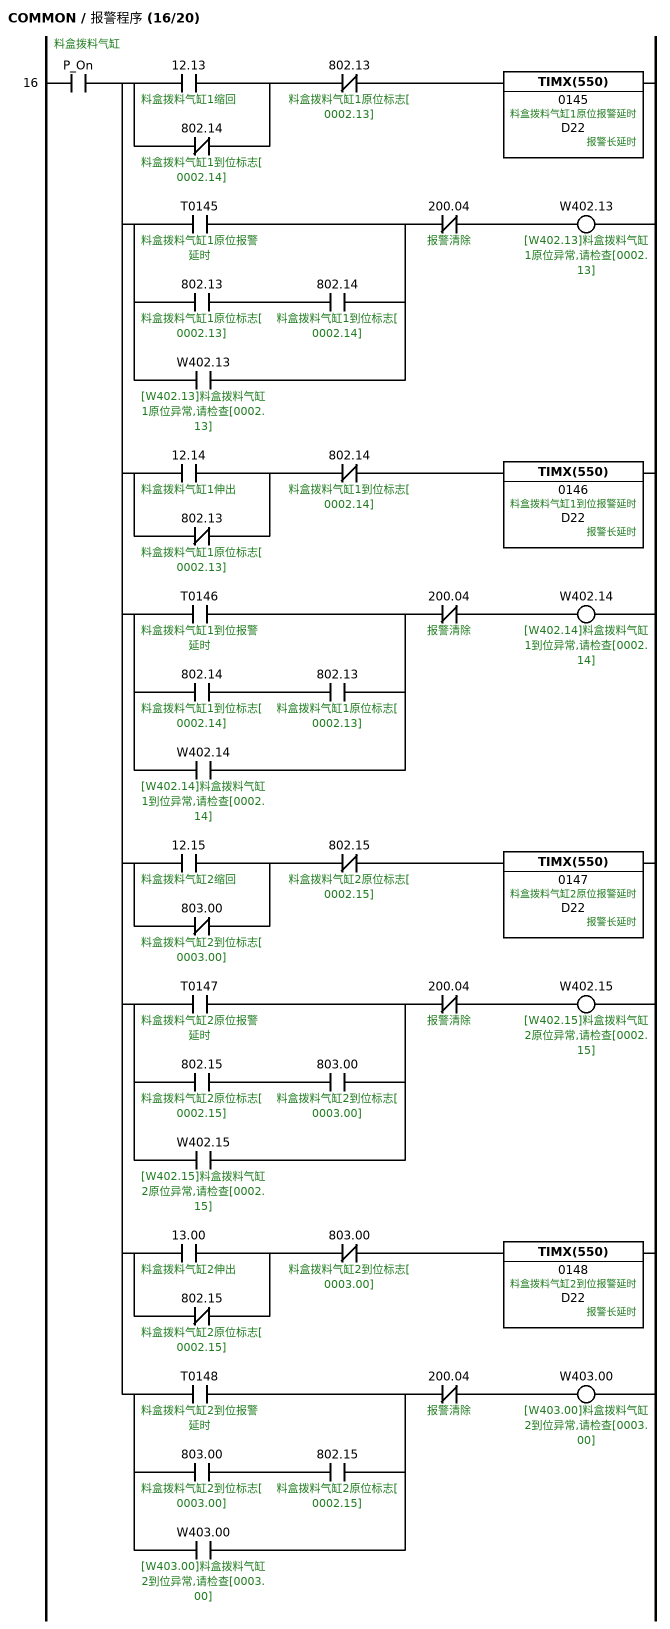
; [picture p192: COMMON / 报警程序, rungs 16-16]
; rung 16: 料盒拨料气缸
LD P_On
OUT TR0
LD 12.13  ; 料盒拨料气缸1缩回
ORNOT 802.14  ; 料盒拨料气缸1到位标志[0002.14]
ANDLD
ANDNOT 802.13  ; 料盒拨料气缸1原位标志[0002.13]
TIMX(550) 0145 D22  ; 报警长延时, 料盒拨料气缸1原位报警延时
LD TR0
LD T0145  ; 料盒拨料气缸1原位报警延时
LD 802.13  ; 料盒拨料气缸1原位标志[0002.13]
AND 802.14  ; 料盒拨料气缸1到位标志[0002.14]
ORLD
OR W402.13  ; [W402.13]料盒拨料气缸1原位异常,请检查[0002.13]
ANDLD
ANDNOT 200.04  ; 报警清除
OUT W402.13  ; [W402.13]料盒拨料气缸1原位异常,请检查[0002.13]
LD TR0
LD 12.14  ; 料盒拨料气缸1伸出
ORNOT 802.13  ; 料盒拨料气缸1原位标志[0002.13]
ANDLD
ANDNOT 802.14  ; 料盒拨料气缸1到位标志[0002.14]
TIMX(550) 0146 D22  ; 报警长延时, 料盒拨料气缸1到位报警延时
LD TR0
LD T0146  ; 料盒拨料气缸1到位报警延时
LD 802.14  ; 料盒拨料气缸1到位标志[0002.14]
AND 802.13  ; 料盒拨料气缸1原位标志[0002.13]
ORLD
OR W402.14  ; [W402.14]料盒拨料气缸1到位异常,请检查[0002.14]
ANDLD
ANDNOT 200.04  ; 报警清除
OUT W402.14  ; [W402.14]料盒拨料气缸1到位异常,请检查[0002.14]
LD TR0
LD 12.15  ; 料盒拨料气缸2缩回
ORNOT 803.00  ; 料盒拨料气缸2到位标志[0003.00]
ANDLD
ANDNOT 802.15  ; 料盒拨料气缸2原位标志[0002.15]
TIMX(550) 0147 D22  ; 报警长延时, 料盒拨料气缸2原位报警延时
LD TR0
LD T0147  ; 料盒拨料气缸2原位报警延时
LD 802.15  ; 料盒拨料气缸2原位标志[0002.15]
AND 803.00  ; 料盒拨料气缸2到位标志[0003.00]
ORLD
OR W402.15  ; [W402.15]料盒拨料气缸2原位异常,请检查[0002.15]
ANDLD
ANDNOT 200.04  ; 报警清除
OUT W402.15  ; [W402.15]料盒拨料气缸2原位异常,请检查[0002.15]
LD TR0
LD 13.00  ; 料盒拨料气缸2伸出
ORNOT 802.15  ; 料盒拨料气缸2原位标志[0002.15]
ANDLD
ANDNOT 803.00  ; 料盒拨料气缸2到位标志[0003.00]
TIMX(550) 0148 D22  ; 报警长延时, 料盒拨料气缸2到位报警延时
LD TR0
LD T0148  ; 料盒拨料气缸2到位报警延时
LD 803.00  ; 料盒拨料气缸2到位标志[0003.00]
AND 802.15  ; 料盒拨料气缸2原位标志[0002.15]
ORLD
OR W403.00  ; [W403.00]料盒拨料气缸2到位异常,请检查[0003.00]
ANDLD
ANDNOT 200.04  ; 报警清除
OUT W403.00  ; [W403.00]料盒拨料气缸2到位异常,请检查[0003.00]

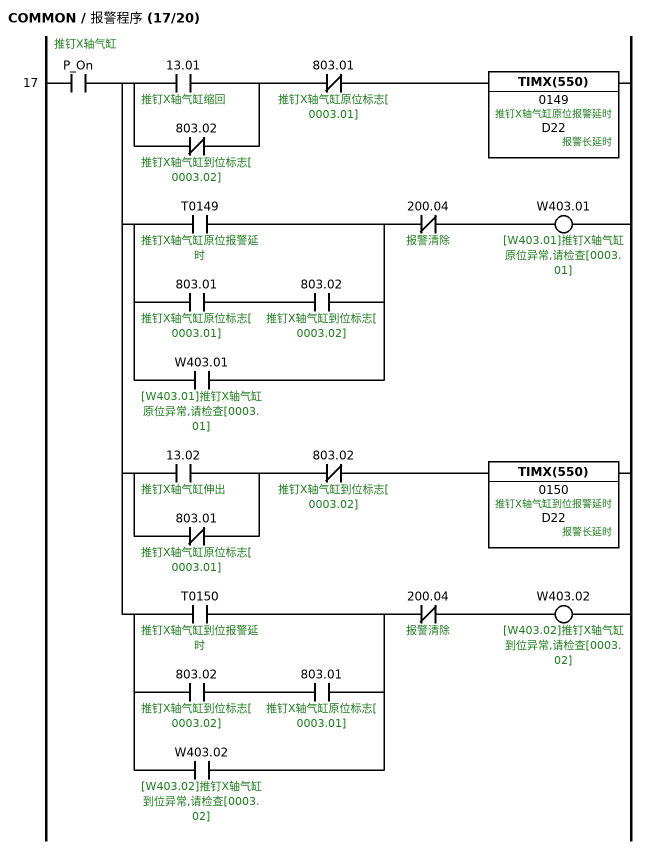
; rung 17: 推钉X轴气缸
LD P_On
OUT TR0
LD 13.01  ; 推钉X轴气缸缩回
ORNOT 803.02  ; 推钉X轴气缸到位标志[0003.02]
ANDLD
ANDNOT 803.01  ; 推钉X轴气缸原位标志[0003.01]
TIMX(550) 0149 D22  ; 报警长延时, 推钉X轴气缸原位报警延时
LD TR0
LD T0149  ; 推钉X轴气缸原位报警延时
LD 803.01  ; 推钉X轴气缸原位标志[0003.01]
AND 803.02  ; 推钉X轴气缸到位标志[0003.02]
ORLD
OR W403.01  ; [W403.01]推钉X轴气缸原位异常,请检查[0003.01]
ANDLD
ANDNOT 200.04  ; 报警清除
OUT W403.01  ; [W403.01]推钉X轴气缸原位异常,请检查[0003.01]
LD TR0
LD 13.02  ; 推钉X轴气缸伸出
ORNOT 803.01  ; 推钉X轴气缸原位标志[0003.01]
ANDLD
ANDNOT 803.02  ; 推钉X轴气缸到位标志[0003.02]
TIMX(550) 0150 D22  ; 报警长延时, 推钉X轴气缸到位报警延时
LD TR0
LD T0150  ; 推钉X轴气缸到位报警延时
LD 803.02  ; 推钉X轴气缸到位标志[0003.02]
AND 803.01  ; 推钉X轴气缸原位标志[0003.01]
ORLD
OR W403.02  ; [W403.02]推钉X轴气缸到位异常,请检查[0003.02]
ANDLD
ANDNOT 200.04  ; 报警清除
OUT W403.02  ; [W403.02]推钉X轴气缸到位异常,请检查[0003.02]

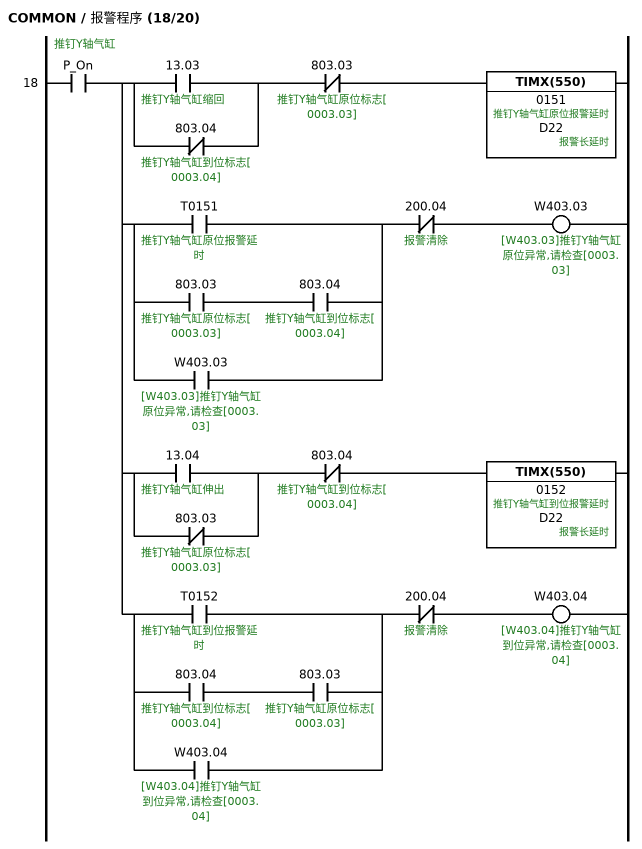
; rung 18: 推钉Y轴气缸
LD P_On
OUT TR0
LD 13.03  ; 推钉Y轴气缸缩回
ORNOT 803.04  ; 推钉Y轴气缸到位标志[0003.04]
ANDLD
ANDNOT 803.03  ; 推钉Y轴气缸原位标志[0003.03]
TIMX(550) 0151 D22  ; 报警长延时, 推钉Y轴气缸原位报警延时
LD TR0
LD T0151  ; 推钉Y轴气缸原位报警延时
LD 803.03  ; 推钉Y轴气缸原位标志[0003.03]
AND 803.04  ; 推钉Y轴气缸到位标志[0003.04]
ORLD
OR W403.03  ; [W403.03]推钉Y轴气缸原位异常,请检查[0003.03]
ANDLD
ANDNOT 200.04  ; 报警清除
OUT W403.03  ; [W403.03]推钉Y轴气缸原位异常,请检查[0003.03]
LD TR0
LD 13.04  ; 推钉Y轴气缸伸出
ORNOT 803.03  ; 推钉Y轴气缸原位标志[0003.03]
ANDLD
ANDNOT 803.04  ; 推钉Y轴气缸到位标志[0003.04]
TIMX(550) 0152 D22  ; 报警长延时, 推钉Y轴气缸到位报警延时
LD TR0
LD T0152  ; 推钉Y轴气缸到位报警延时
LD 803.04  ; 推钉Y轴气缸到位标志[0003.04]
AND 803.03  ; 推钉Y轴气缸原位标志[0003.03]
ORLD
OR W403.04  ; [W403.04]推钉Y轴气缸到位异常,请检查[0003.04]
ANDLD
ANDNOT 200.04  ; 报警清除
OUT W403.04  ; [W403.04]推钉Y轴气缸到位异常,请检查[0003.04]

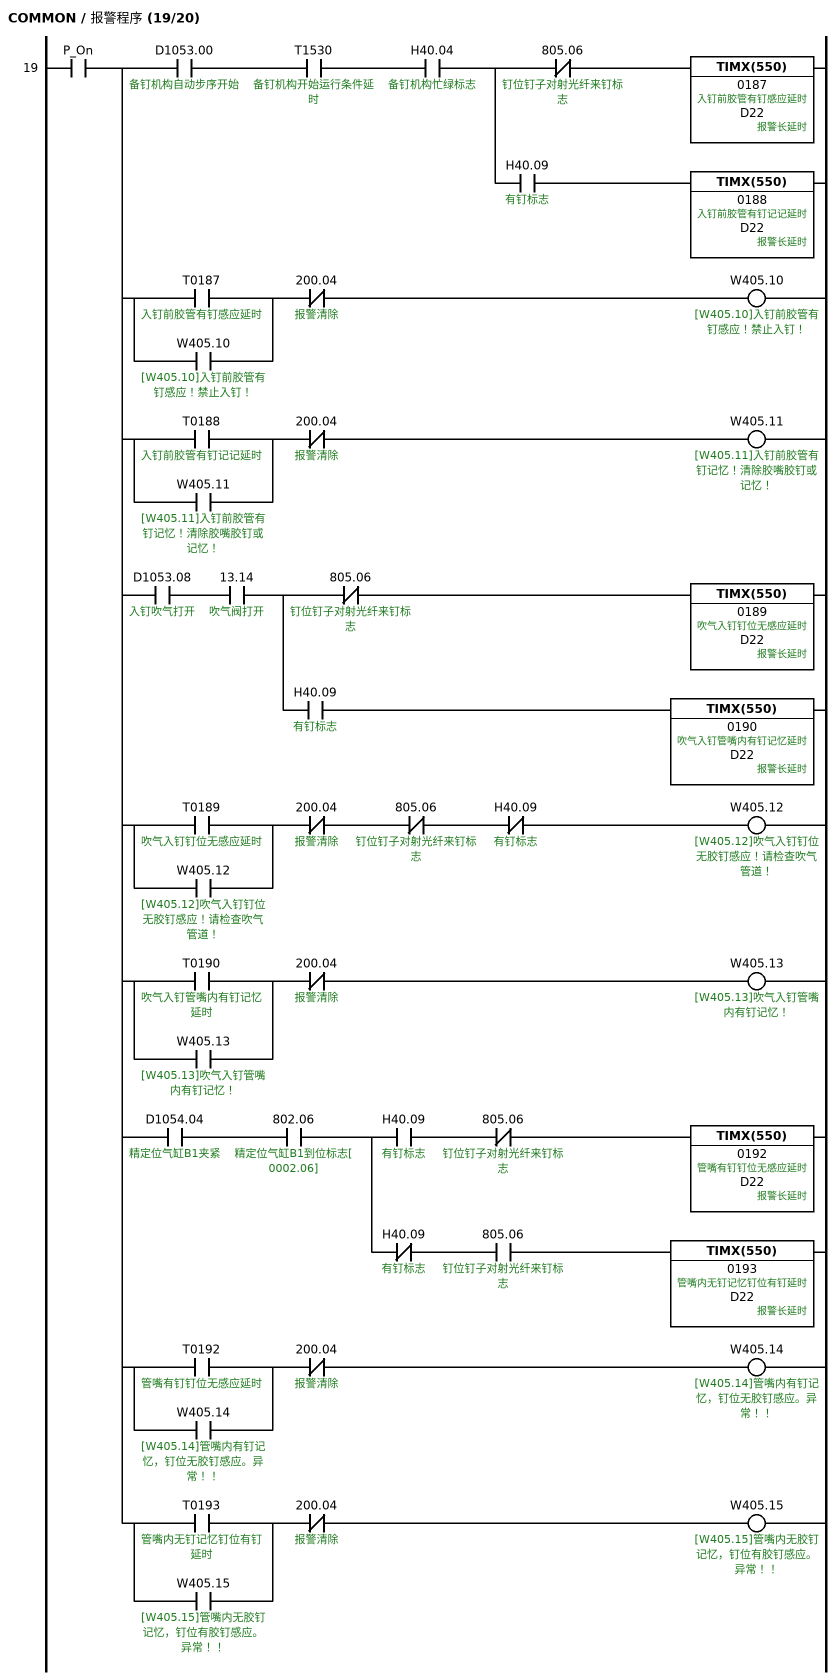
; rung 19
LD P_On
OUT TR0
AND D1053.00  ; 备钉机构自动步序开始
AND T1530  ; 备钉机构开始运行条件延时
AND H40.04  ; 备钉机构忙绿标志
OUT TR1
ANDNOT 805.06  ; 钉位钉子对射光纤来钉标志
TIMX(550) 0187 D22  ; 报警长延时, 入钉前胶管有钉感应延时
LD TR1
AND H40.09  ; 有钉标志
TIMX(550) 0188 D22  ; 报警长延时, 入钉前胶管有钉记记延时
LD TR0
LD T0187  ; 入钉前胶管有钉感应延时
OR W405.10  ; [W405.10]入钉前胶管有钉感应！禁止入钉！
ANDLD
ANDNOT 200.04  ; 报警清除
OUT W405.10  ; [W405.10]入钉前胶管有钉感应！禁止入钉！
LD TR0
LD T0188  ; 入钉前胶管有钉记记延时
OR W405.11  ; [W405.11]入钉前胶管有钉记忆！清除胶嘴胶钉或记忆！
ANDLD
ANDNOT 200.04  ; 报警清除
OUT W405.11  ; [W405.11]入钉前胶管有钉记忆！清除胶嘴胶钉或记忆！
LD TR0
AND D1053.08  ; 入钉吹气打开
AND 13.14  ; 吹气阀打开
OUT TR1
ANDNOT 805.06  ; 钉位钉子对射光纤来钉标志
TIMX(550) 0189 D22  ; 报警长延时, 吹气入钉钉位无感应延时
LD TR1
AND H40.09  ; 有钉标志
TIMX(550) 0190 D22  ; 报警长延时, 吹气入钉管嘴内有钉记忆延时
LD TR0
LD T0189  ; 吹气入钉钉位无感应延时
OR W405.12  ; [W405.12]吹气入钉钉位无胶钉感应！请检查吹气管道！
ANDLD
ANDNOT 200.04  ; 报警清除
ANDNOT 805.06  ; 钉位钉子对射光纤来钉标志
ANDNOT H40.09  ; 有钉标志
OUT W405.12  ; [W405.12]吹气入钉钉位无胶钉感应！请检查吹气管道！
LD TR0
LD T0190  ; 吹气入钉管嘴内有钉记忆延时
OR W405.13  ; [W405.13]吹气入钉管嘴内有钉记忆！
ANDLD
ANDNOT 200.04  ; 报警清除
OUT W405.13  ; [W405.13]吹气入钉管嘴内有钉记忆！
LD TR0
AND D1054.04  ; 精定位气缸B1夹紧
AND 802.06  ; 精定位气缸B1到位标志[0002.06]
OUT TR1
AND H40.09  ; 有钉标志
ANDNOT 805.06  ; 钉位钉子对射光纤来钉标志
TIMX(550) 0192 D22  ; 报警长延时, 管嘴有钉钉位无感应延时
LD TR1
ANDNOT H40.09  ; 有钉标志
AND 805.06  ; 钉位钉子对射光纤来钉标志
TIMX(550) 0193 D22  ; 报警长延时, 管嘴内无钉记忆钉位有钉延时
LD TR0
LD T0192  ; 管嘴有钉钉位无感应延时
OR W405.14  ; [W405.14]管嘴内有钉记忆，钉位无胶钉感应。异常！！
ANDLD
ANDNOT 200.04  ; 报警清除
OUT W405.14  ; [W405.14]管嘴内有钉记忆，钉位无胶钉感应。异常！！
LD TR0
LD T0193  ; 管嘴内无钉记忆钉位有钉延时
OR W405.15  ; [W405.15]管嘴内无胶钉记忆，钉位有胶钉感应。异常！！
ANDLD
ANDNOT 200.04  ; 报警清除
OUT W405.15  ; [W405.15]管嘴内无胶钉记忆，钉位有胶钉感应。异常！！

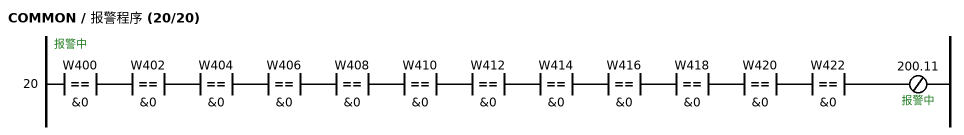
; rung 20: 报警中
LD=L(301) W400 &0
AND=L(301) W402 &0
AND=L(301) W404 &0
AND=L(301) W406 &0
AND=L(301) W408 &0
AND=L(301) W410 &0
AND=L(301) W412 &0
AND=L(301) W414 &0
AND=L(301) W416 &0
AND=L(301) W418 &0
AND=L(301) W420 &0
AND=(300) W422 &0
OUTNOT 200.11  ; 报警中

### Section PC交互

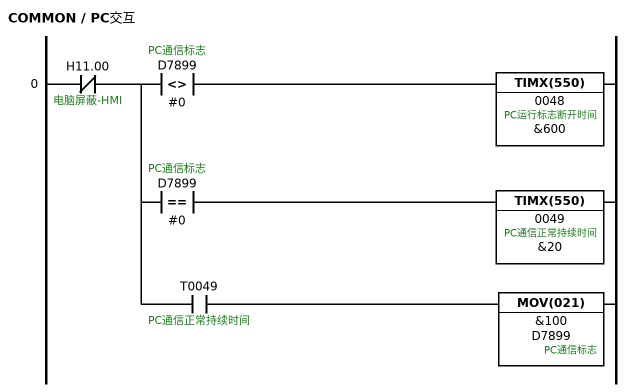
; rung 0
LDNOT H11.00  ; 电脑屏蔽-HMI
OUT TR0
AND<>(305) D7899 #0  ; PC通信标志
TIMX(550) 0048 &600  ; PC运行标志断开时间
LD TR0
AND=(300) D7899 #0  ; PC通信标志
TIMX(550) 0049 &20  ; PC通信正常持续时间
LD TR0
AND T0049  ; PC通信正常持续时间
MOV(021) &100 D7899  ; PC通信标志

### Section END
; rung 0
END(001)